Staubli VAL3: getAction.pgx

public program getAction(ActionItem& x_aAction (dimensions=1))
begin
  // mutex it
  setMutex(bActionMutex)
  // give back the action on first element
  x_aAction=aAction[0]
  //release
  bActionMutex=false
end
